PROGRAM MAIN
VAR
END_VAR


CraneSimulation();


//IF Inputs.bStart THEN
//	Outputs.bSimRunning := TRUE;
//	ELSE
//		Outputs.bSimRunning := FALSE;
//END_IF

END_PROGRAM

(* stored: Version 1.1.0.1, ProductVersion 3.1.4024.10
   POU MAIN: Id {2bcbf739-3111-45d7-9a18-ef40f2d3cd09}, SpecialFunc None *)
